// TIA Portal V19 export
TYPE "LAF_typeInterfaceSignalsBool"
TITLE = Interface signals bool / PLC_DIAG
// The data structure for the interface bool functionality. The type contains all relevant information for one interface bool function block.
// 
// **PLC Data types**  
// * [LAF_typeInterfaceSignals](../Library%20Types/LAF_typeInterfaceSignals.htm)
// Struktur Schnittstellen Signale
// stored: Access Published
   STRUCT
      readValue { ExternalAccessible := 'False'; ExternalVisible := 'False'; ExternalWritable := 'False'} : Bool;   // Zustand der Signale zyklisch aktualisieren / Refresh state of signals cyclic
      readSymbolicName { ExternalAccessible := 'False'; ExternalVisible := 'False'; ExternalWritable := 'False'} : Bool;   // Einmaliges neues Einlesen der Symbolischen Namen / Read symbolic name (again)
      freeDescriptionText : WString[40] := WSTRING#'Click on the pencil to enter description';   // HMI: Freier zu vergebender Text / HMI: Free text for description
      interfaceSignalBool : Array[0..15] of "LAF_typeInterfaceSignals";   // HMI: Wert und Symbolischer Name / HMI: Value and symbolic name
   END_STRUCT;
END_TYPE
